TYPE ParIDAccess_Status_axis_typ :
	STRUCT	
		WriteCoeSdo			: ParIDAccess_Status_typ ;
		ReadCoeSdo			: ParIDAccess_Status_typ ;	
	END_STRUCT
END_TYPE

(* stored: Version 1.1.0.1, ProductVersion 3.1.4024.3
   DUT ParIDAccess_Status_axis_typ: Id {a8fdd55d-2a95-0bff-3060-1938d6188ebf} *)
